// TIA Portal V18 export
DATA_BLOCK "air_data"   // DB1
{ S7_Optimized_Access := 'TRUE' }
VERSION : 0.1
// stored: AutoNumber true, DBAccessibleFromOPCUA true, IsOnlyStoredInLoadMemory false, IsRetainMemResEnabled false, IsWriteProtectedInAS false, MemoryReserve 100
   VAR RETAIN
      calc_const { S7_SetPoint := 'True'} : "quad_cnst_array";
      Pmean { S7_SetPoint := 'True'} : Real := 1013.25;   // Mean atmospheric pressure [hPa] (mbar)
   END_VAR
BEGIN
END_DATA_BLOCK
